DATA_BLOCK "DB"
{ S7_Optimized_Access := 'false' }
    VAR
        i: DINT;
        bol: BOOL;
        col: BYTE;
        aut_y: REAL;
        firstRun: BOOL;
    END_VAR
BEGIN
    firstRun := TRUE;
END_DATA_BLOCK
